// TwinCAT 3 PLC project TypesTests
// ProgramVersion: 3.1.4024.0
// libraries:
//   Tc2_Standard, * (Beckhoff Automation GmbH)
//   Tc2_System, * (Beckhoff Automation GmbH)
//   Tc3_Module, * (Beckhoff Automation GmbH)
//   TcUnit, * (www.tcunit.org)
//   Types, * (TomasRompotl)
// project tree:
//   / PlcTask.TcTTO
//   Tests/Any/ AnyTypeTest.TcPOU
//   Tests/Binding/ BindTest.TcPOU, NotBindTest.TcPOU, BoolBindingReadOnlyTest.TcPOU
//   Tests/ PRG_Test.TcPOU
//   Tests/Values/BooleanExpression/ BooleanExpressionTest.TcPOU, BooleanExpressionFunctionsTest.TcPOU
//   Tests/_TemplateTest/ _TemplateTest.TcPOU
//   Tests/Reflection/ ReflectionTest.TcPOU
//   Tests/Values/ BoolValuesTest.TcPOU

CONFIGURATION TypesTests
    RESOURCE PLC ON TwinCAT3
        TASK PlcTask(INTERVAL := T#1ms, PRIORITY := 20);
        PROGRAM PRG_Test WITH PlcTask : PRG_Test;
    END_RESOURCE
END_CONFIGURATION

// ---- Tests/PRG_Test.TcPOU
PROGRAM PRG_Test
VAR
	anyTypeBindedTest : AnyTypeTest;
	boolBindingReadOnlyTest : BoolBindingReadOnlyTest;
	bindTest : BindTest;
	notBindTest : NotBindTest;
	
	reflectionTest : ReflectionTest;
	
	boolValuesTest : BoolValuesTest;
	booleanExpressionTest : BooleanExpressionTest;
	booleanExpressionFunctionsTest : BooleanExpressionFunctionsTest;
END_VAR

TcUnit.RUN();

END_PROGRAM

// ---- Tests/Any/AnyTypeTest.TcPOU
FUNCTION_BLOCK AnyTypeTest EXTENDS TcUnit.FB_TestSuite

CheckIsAnyTypeBinded();
ToAnyTypeFunction();

METHOD CheckIsAnyTypeBinded 
VAR
	isOpen : BOOL;
	nonBound : __SYSTEM.AnyType; 
END_VAR
TcUnit.TEST('Check is any type bounded');

AssertEquals_BOOL(
	Expected := FALSE,
	Actual   := isAnyTypeBinded(anyType := nonBound),
	Message  := 'Expected FALSE when anyType is not bounded');

AssertEquals_BOOL(
	Expected := TRUE,
	Actual   := isAnyTypeBinded(anyType := ToAnyType(isOpen)),
	Message  := 'Expected TRUE when anyType is bounded');

TEST_FINISHED();
END_METHOD

METHOD ToAnyTypeFunction
VAR  
	intValue : INT;
	returnOfAnyType : __SYSTEM.AnyType;
	pIntValue : POINTER TO INT;
END_VAR
TcUnit.TEST('To AnyType Function');

returnOfAnyType := ToAnyType(intValue);
pIntValue := ADR(intValue);

AssertEquals(
	Expected := pIntValue,
	Actual   := returnOfAnyType.pValue,
	Message  := 'ToAnyType() failed: pValue was 0 or diSize was incorrect for int input.');

TEST_FINISHED();
END_METHOD

END_FUNCTION_BLOCK

// ---- Tests/Binding/BoolBindingReadOnlyTest.TcPOU
FUNCTION_BLOCK BoolBindingReadOnlyTest EXTENDS TcUnit.FB_TestSuite

CheckIsBinded();
BindingReturnsSameValue();
NegatedBindingReturnsNegatedValue();

METHOD BindingReturnsSameValue : BOOL
VAR
	expected : BOOL;
	actual : BOOL;
	
	binding : BoolBindingReadOnly;
	variable : BOOL;
END_VAR
TcUnit.TEST('Binding returns same value');

binding.Bind(variable);

expected := FALSE;
actual := binding.Value;

AssertEquals(
	Expected := expected,
	Actual := actual,
	Message := 'Value should return FALSE if binded variable is FALSE');
	
variable := TRUE;

expected := TRUE;
actual := binding.Value;

AssertEquals(
	Expected := expected,
	Actual := actual,
	Message := 'Value should return TRUE if binded variable is TRUE');

TEST_FINISHED();
END_METHOD

METHOD CheckIsBinded : BOOL
VAR
	expected : BOOL;
	actual : BOOL;
	
	binding : BoolBindingReadOnly;
	variable : BOOL;
END_VAR
TcUnit.TEST('Check binded');

expected := FALSE;
actual := binding.IsBinded;

AssertEquals(
	Expected := expected,
	Actual := actual,
	Message := 'IsBinded should be FALSE before binding');

binding.Bind(variable);

expected := TRUE;
actual := binding.IsBinded;

AssertEquals(
	Expected := expected,
	Actual := actual,
	Message := 'IsBinded should be TRUE after successful Bind()');

TEST_FINISHED();
END_METHOD

METHOD NegatedBindingReturnsNegatedValue : BOOL
VAR
	expected : BOOL;
	actual : BOOL;
	
	binding : BoolBindingReadOnly;
	variable : BOOL;
END_VAR
TcUnit.TEST('Negated binding returns negated value');

binding.Bind(variable);
binding.Negate := TRUE;

expected := TRUE;
actual := binding.Value;

AssertEquals(
	Expected := expected,
	Actual := actual,
	Message := 'Value should return TRUE if binded variable is FALSE');
	
variable := TRUE;

expected := FALSE;
actual := binding.Value;

AssertEquals(
	Expected := expected,
	Actual := actual,
	Message := 'Value should return FALSE if binded variable is TRUE');

TEST_FINISHED();
END_METHOD

END_FUNCTION_BLOCK

// ---- Tests/Binding/BindTest.TcPOU
FUNCTION_BLOCK BindTest EXTENDS TcUnit.FB_TestSuite

BindAndTestBinding();

METHOD BindAndTestBinding : BOOL
VAR
	expected : BOOL;
	actual : BOOL;
	
	variable : BOOL;
	binding : BoolValue;
	disposable : Disposable;
END_VAR
TcUnit.TEST('Bind and test binding');

binding := Bind(variable);

expected := TRUE;
actual := binding <> 0;

AssertEquals(
	Expected := expected,
	Actual := actual,
	Message := 'Bind should return interface to created Binding');
	
variable := TRUE;

expected := TRUE;
actual := binding.Value;

AssertEquals(
	Expected := expected,
	Actual := actual,
	Message := 'Binding should return value of binded variable');
	
__QUERYINTERFACE(binding, disposable);
disposable.Dispose();

TEST_FINISHED();
END_METHOD

END_FUNCTION_BLOCK

// ---- Tests/Binding/NotBindTest.TcPOU
FUNCTION_BLOCK NotBindTest EXTENDS TcUnit.FB_TestSuite

BindAndTestBinding();

METHOD BindAndTestBinding : BOOL
VAR
	expected : BOOL;
	actual : BOOL;
	
	variable : BOOL;
	binding : BoolValue;
	disposable : Disposable;
END_VAR
TcUnit.TEST('Bind and test binding');

binding := NotBind(variable);

expected := TRUE;
actual := binding <> 0;

AssertEquals(
	Expected := expected,
	Actual := actual,
	Message := 'NotBind should return interface to created Binding');
	
variable := FALSE;

expected := TRUE;
actual := binding.Value;

AssertEquals(
	Expected := expected,
	Actual := actual,
	Message := 'Binding should return negated value of binded variable');
	
__QUERYINTERFACE(binding, disposable);
disposable.Dispose();

TEST_FINISHED();
END_METHOD

END_FUNCTION_BLOCK

// ---- Tests/Reflection/ReflectionTest.TcPOU
FUNCTION_BLOCK ReflectionTest EXTENDS TcUnit.FB_TestSuite
VAR
	reflection : Reflection(THIS, SIZEOF(THIS^));
END_VAR

GetAllData();

METHOD GetAllData : BOOL
VAR
END_VAR
TcUnit.TEST('Get all data');

AssertEquals_STRING(
	Actual := reflection.InstanceName,
	Expected := 'FrameworkMonorepo.TypesTests.PRG_Test.reflectionTest',
	Message := 'InstanceName was not obtained correctly');

AssertEquals_STRING(
	Actual := reflection.SolutionName,
	Expected := 'FrameworkMonorepo',
	Message := 'SolutionName was not obtained correctly');

AssertEquals_STRING(
	Actual := reflection.ProjectName,
	Expected := 'TypesTests',
	Message := 'ProjectName was not obtained correctly');

AssertEquals_STRING(
	Actual := reflection.ParentName,
	Expected := 'PRG_Test',
	Message := 'ParentName was not obtained correctly');

AssertEquals_STRING(
	Actual := reflection.Name,
	Expected := 'reflectionTest',
	Message := 'Name was not obtained correctly');

AssertEquals_STRING(
	Actual := reflection.ObjectPath,
	Expected := 'PRG_Test.reflectionTest',
	Message := 'ObjectPath was not obtained correctly');

AssertEquals_STRING(
	Actual := reflection.TypeName,
	Expected := 'ReflectionTest',
	Message := 'TypeName was not obtained correctly');

TEST_FINISHED();
END_METHOD

END_FUNCTION_BLOCK

// ---- Tests/Values/BoolValuesTest.TcPOU
FUNCTION_BLOCK BoolValuesTest EXTENDS TcUnit.FB_TestSuite

FalseBoolValue();
TrueBoolValue();

METHOD FalseBoolValue : BOOL
VAR
	value : FalseBoolValue;
END_VAR
TcUnit.TEST('Get false bool value');

AssertEquals_BOOL(
	Expected := FALSE,
	Actual := value.Value,
	Message := 'FalseBoolValue should return FALSE value');

TEST_FINISHED();
END_METHOD

METHOD TrueBoolValue : BOOL
VAR
	value : TrueBoolValue;
END_VAR
TcUnit.TEST('Get true bool value');

AssertEquals_BOOL(
	Expected := TRUE,
	Actual := value.Value,
	Message := 'TrueBoolValue should return TRUE value');

TEST_FINISHED();
END_METHOD

END_FUNCTION_BLOCK

// ---- Tests/Values/BooleanExpression/BooleanExpressionTest.TcPOU
FUNCTION_BLOCK BooleanExpressionTest EXTENDS TcUnit.FB_TestSuite

Bind2Operands();

METHOD Bind2Operands : BOOL
VAR
	val1 : BOOL;
	val2 : BOOL;
	expAnd : BooleanExpression;
	expOr : BooleanExpression;
	expXor : BooleanExpression;
END_VAR
TcUnit.TEST('Bind 2 operands');

expAnd.Op2(BooleanOperator.ANDop, Bind(val1), Bind(val2));
expOr.Op2(BooleanOperator.ORop, Bind(val1), Bind(val2));
expXor.Op2(BooleanOperator.XORop, Bind(val1), Bind(val2));

val1 := FALSE;
val2 := FALSE;

AssertEquals_BOOL(
	Expected := FALSE,
	Actual := expAnd.Value,
	Message := 'FALSE AND FALSE should be FALSE');
AssertEquals_BOOL(
	Expected := FALSE,
	Actual := expOr.Value,
	Message := 'FALSE OR FALSE should be FALSE');
AssertEquals_BOOL(
	Expected := FALSE,
	Actual := expXor.Value,
	Message := 'FALSE XOR FALSE should be FALSE');

val1 := TRUE;
val2 := FALSE;

AssertEquals_BOOL(
	Expected := FALSE,
	Actual := expAnd.Value,
	Message := 'TRUE AND FALSE should be FALSE');
AssertEquals_BOOL(
	Expected := TRUE,
	Actual := expOr.Value,
	Message := 'TRUE OR FALSE should be TRUE');
AssertEquals_BOOL(
	Expected := TRUE,
	Actual := expXor.Value,
	Message := 'TRUE XOR FALSE should be TRUE');

val1 := TRUE;
val2 := TRUE;

AssertEquals_BOOL(
	Expected := TRUE,
	Actual := expAnd.Value,
	Message := 'TRUE AND TRUE should be TRUE');
AssertEquals_BOOL(
	Expected := TRUE,
	Actual := expOr.Value,
	Message := 'TRUE OR TRUE should be TRUE');
AssertEquals_BOOL(
	Expected := FALSE,
	Actual := expXor.Value,
	Message := 'TRUE XOR TRUE should be FALSE');

TEST_FINISHED();
END_METHOD

END_FUNCTION_BLOCK

// ---- Tests/Values/BooleanExpression/BooleanExpressionFunctionsTest.TcPOU
FUNCTION_BLOCK BooleanExpressionFunctionsTest EXTENDS TcUnit.FB_TestSuite

And234();
Or234();
Xor234();

METHOD And234 : BOOL
VAR
	bool1 : BOOL;
	bool2 : BOOL;
	bool3 : BOOL;
	bool4 : BOOL;
	value2 : BoolValue;
	value3 : BoolValue;
	value4 : BoolValue;
	disposable : Disposable;
END_VAR
TcUnit.TEST('Functions And2, 3, 4');

value2 := And2(Bind(bool1), Bind(bool2));
value3 := And3(Bind(bool1), Bind(bool2), Bind(bool3));
value4 := And4(Bind(bool1), Bind(bool2), Bind(bool3), Bind(bool4));

bool1 := FALSE;
bool2 := FALSE;
bool3 := FALSE;
bool4 := FALSE;

AssertEquals_BOOL(
	Expected := FALSE,
	Actual := value2.Value,
	Message := 'FALSE AND FALSE should be FALSE');
AssertEquals_BOOL(
	Expected := FALSE,
	Actual := value3.Value,
	Message := 'FALSE AND FALSE AND FALSE should be FALSE');
AssertEquals_BOOL(
	Expected := FALSE,
	Actual := value4.Value,
	Message := 'FALSE AND FALSE AND FALSE AND FALSE should be FALSE');

bool1 := TRUE;
bool2 := FALSE;
bool3 := FALSE;
bool4 := FALSE;

AssertEquals_BOOL(
	Expected := FALSE,
	Actual := value2.Value,
	Message := 'TRUE AND FALSE should be FALSE');
AssertEquals_BOOL(
	Expected := FALSE,
	Actual := value3.Value,
	Message := 'TRUE AND FALSE AND FALSE should be FALSE');
AssertEquals_BOOL(
	Expected := FALSE,
	Actual := value4.Value,
	Message := 'TRUE AND FALSE AND FALSE AND FALSE should be FALSE');

bool1 := TRUE;
bool2 := TRUE;
bool3 := TRUE;
bool4 := TRUE;

AssertEquals_BOOL(
	Expected := TRUE,
	Actual := value2.Value,
	Message := 'TRUE AND TRUE should be TRUE');
AssertEquals_BOOL(
	Expected := TRUE,
	Actual := value3.Value,
	Message := 'TRUE AND TRUE AND TRUE should be TRUE');
AssertEquals_BOOL(
	Expected := TRUE,
	Actual := value4.Value,
	Message := 'TRUE AND TRUE AND TRUE AND TRUE should be TRUE');

__QUERYINTERFACE(value2, disposable);
disposable.Dispose();
__QUERYINTERFACE(value3, disposable);
disposable.Dispose();
__QUERYINTERFACE(value4, disposable);
disposable.Dispose();

TEST_FINISHED();
END_METHOD

METHOD Or234 : BOOL
VAR
	bool1 : BOOL;
	bool2 : BOOL;
	bool3 : BOOL;
	bool4 : BOOL;
	value2 : BoolValue;
	value3 : BoolValue;
	value4 : BoolValue;
	disposable : Disposable;
END_VAR
TcUnit.TEST('Functions Or2, 3, 4');

value2 := Or2(Bind(bool1), Bind(bool2));
value3 := Or3(Bind(bool1), Bind(bool2), Bind(bool3));
value4 := Or4(Bind(bool1), Bind(bool2), Bind(bool3), Bind(bool4));

bool1 := FALSE;
bool2 := FALSE;
bool3 := FALSE;
bool4 := FALSE;

AssertEquals_BOOL(
	Expected := FALSE,
	Actual := value2.Value,
	Message := 'FALSE OR FALSE should be FALSE');
AssertEquals_BOOL(
	Expected := FALSE,
	Actual := value3.Value,
	Message := 'FALSE OR FALSE OR FALSE should be FALSE');
AssertEquals_BOOL(
	Expected := FALSE,
	Actual := value4.Value,
	Message := 'FALSE OR FALSE OR FALSE OR FALSE should be FALSE');

bool1 := TRUE;
bool2 := FALSE;
bool3 := FALSE;
bool4 := FALSE;

AssertEquals_BOOL(
	Expected := TRUE,
	Actual := value2.Value,
	Message := 'TRUE OR FALSE should be TRUE');
AssertEquals_BOOL(
	Expected := TRUE,
	Actual := value3.Value,
	Message := 'TRUE OR FALSE OR FALSE should be TRUE');
AssertEquals_BOOL(
	Expected := TRUE,
	Actual := value4.Value,
	Message := 'TRUE OR FALSE OR FALSE OR FALSE should be TRUE');

bool1 := TRUE;
bool2 := TRUE;
bool3 := TRUE;
bool4 := TRUE;

AssertEquals_BOOL(
	Expected := TRUE,
	Actual := value2.Value,
	Message := 'TRUE OR TRUE should be TRUE');
AssertEquals_BOOL(
	Expected := TRUE,
	Actual := value3.Value,
	Message := 'TRUE OR TRUE OR TRUE should be TRUE');
AssertEquals_BOOL(
	Expected := TRUE,
	Actual := value4.Value,
	Message := 'TRUE OR TRUE OR TRUE OR TRUE should be TRUE');

__QUERYINTERFACE(value2, disposable);
disposable.Dispose();
__QUERYINTERFACE(value3, disposable);
disposable.Dispose();
__QUERYINTERFACE(value4, disposable);
disposable.Dispose();

TEST_FINISHED();
END_METHOD

METHOD Xor234 : BOOL
VAR
	bool1 : BOOL;
	bool2 : BOOL;
	bool3 : BOOL;
	bool4 : BOOL;
	value2 : BoolValue;
	value3 : BoolValue;
	value4 : BoolValue;
	disposable : Disposable;
END_VAR
TcUnit.TEST('Functions Xor2, 3, 4');

value2 := Xor2(Bind(bool1), Bind(bool2));
value3 := Xor3(Bind(bool1), Bind(bool2), Bind(bool3));
value4 := Xor4(Bind(bool1), Bind(bool2), Bind(bool3), Bind(bool4));

bool1 := FALSE;
bool2 := FALSE;
bool3 := FALSE;
bool4 := FALSE;

AssertEquals_BOOL(
	Expected := FALSE,
	Actual := value2.Value,
	Message := 'FALSE XOR FALSE should be FALSE');
AssertEquals_BOOL(
	Expected := FALSE,
	Actual := value3.Value,
	Message := 'FALSE XOR FALSE XOR FALSE should be FALSE');
AssertEquals_BOOL(
	Expected := FALSE,
	Actual := value4.Value,
	Message := 'FALSE XOR FALSE XOR FALSE XOR FALSE should be FALSE');

bool1 := TRUE;
bool2 := FALSE;
bool3 := FALSE;
bool4 := FALSE;

AssertEquals_BOOL(
	Expected := TRUE,
	Actual := value2.Value,
	Message := 'TRUE XOR FALSE should be TRUE');
AssertEquals_BOOL(
	Expected := TRUE,
	Actual := value3.Value,
	Message := 'TRUE XOR FALSE XOR FALSE should be TRUE');
AssertEquals_BOOL(
	Expected := TRUE,
	Actual := value4.Value,
	Message := 'TRUE XOR FALSE XOR FALSE XOR FALSE should be TRUE');

bool1 := TRUE;
bool2 := TRUE;
bool3 := TRUE;
bool4 := TRUE;

AssertEquals_BOOL(
	Expected := FALSE,
	Actual := value2.Value,
	Message := 'TRUE XOR TRUE should be FALSE');
AssertEquals_BOOL(
	Expected := TRUE,
	Actual := value3.Value,
	Message := 'TRUE XOR TRUE XOR TRUE should be TRUE');
AssertEquals_BOOL(
	Expected := FALSE,
	Actual := value4.Value,
	Message := 'TRUE XOR TRUE XOR TRUE XOR TRUE should be FALSE');

__QUERYINTERFACE(value2, disposable);
disposable.Dispose();
__QUERYINTERFACE(value3, disposable);
disposable.Dispose();
__QUERYINTERFACE(value4, disposable);
disposable.Dispose();

TEST_FINISHED();
END_METHOD

END_FUNCTION_BLOCK

// ---- Tests/_TemplateTest/_TemplateTest.TcPOU
FUNCTION_BLOCK _TemplateTest EXTENDS TcUnit.FB_TestSuite
VAR
END_VAR

ExampleTest();

METHOD ExampleTest : BOOL
VAR
	expected : INT;
	actual : INT;
END_VAR
TcUnit.TEST('Example test');

expected := ;
actual := ;

AssertEquals(
	Expected := expected,
	Actual := actual,
	Message := 'What went wrong');

TEST_FINISHED();
END_METHOD

END_FUNCTION_BLOCK
